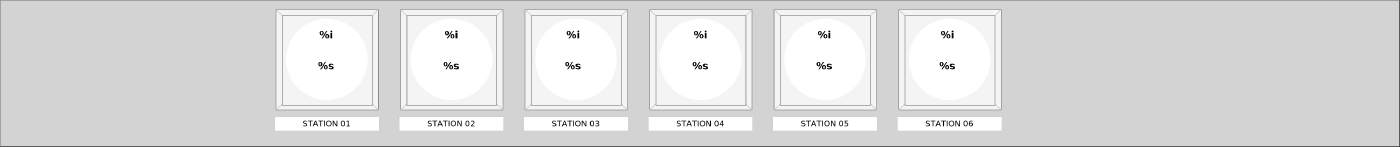
VISUALIZATION Popup_ProcessStatus  // 2001x211
    Rectangle (0,0 2001x211)
    Group (570,13 150x175)
        RoundedRectangle (0,154 150x21), "STATION 02"
        Image (2,0 147x145)
            p573394764: StartStop.Value
        Pie (11,9 129x129)
            p426801730: iDisplayTimeCycle[2]
            p2124672552: iDisplayTimeCycleEnd[2]
        Ellipse (17,14 116x116), colour toggle: bDisplayTimeCycleOn[2]
        Rectangle (29,42 92x79), "%s", text variable: ARsStnProcessName[2]
        Rectangle (41,22 69x30), "%i", text variable: ARiStnProcessTimeCD[2]
    Group (392,13 150x175)
        RoundedRectangle (0,154 150x21), "STATION 01"
        Image (2,0 147x145)
            p573394764: StartStop.Value
        Pie (11,9 129x129)
            p426801730: iDisplayTimeCycle[1]
            p2124672552: iDisplayTimeCycleEnd[1]
        Ellipse (17,14 116x116), colour toggle: bDisplayTimeCycleOn[1]
        Rectangle (28,42 92x79), "%s", text variable: ARsStnProcessName[1]
        Rectangle (40,22 69x30), "%i", text variable: ARiStnProcessTimeCD[1]
    Group (748,13 150x175)
        RoundedRectangle (0,154 150x21), "STATION 03"
        Image (2,0 147x145)
            p573394764: StartStop.Value
        Pie (11,9 129x129)
            p426801730: iDisplayTimeCycle[3]
            p2124672552: iDisplayTimeCycleEnd[3]
        Ellipse (17,14 116x116), colour toggle: bDisplayTimeCycleOn[3]
        Rectangle (25,42 92x79), "%s", text variable: ARsStnProcessName[3]
        Rectangle (37,22 69x30), "%i", text variable: ARiStnProcessTimeCD[3]
    Group (926,13 150x175)
        RoundedRectangle (0,154 150x21), "STATION 04"
        Image (2,0 147x145)
            p573394764: StartStop.Value
        Pie (11,9 129x129)
            p426801730: iDisplayTimeCycle[4]
            p2124672552: iDisplayTimeCycleEnd[4]
        Ellipse (17,14 116x116), colour toggle: bDisplayTimeCycleOn[4]
        Rectangle (29,42 92x79), "%s", text variable: ARsStnProcessName[4]
        Rectangle (41,22 69x30), "%i", text variable: ARiStnProcessTimeCD[4]
    Group (1104,13 150x175)
        RoundedRectangle (0,154 150x21), "STATION 05"
        Image (2,0 147x145)
            p573394764: StartStop.Value
        Pie (11,9 129x129)
            p426801730: iDisplayTimeCycle[5]
            p2124672552: iDisplayTimeCycleEnd[5]
        Ellipse (17,14 116x116), colour toggle: bDisplayTimeCycleOn[5]
        Rectangle (28,42 92x79), "%s", text variable: ARsStnProcessName[5]
        Rectangle (40,22 69x30), "%i", text variable: ARiStnProcessTimeCD[5]
    Group (1282,13 150x175)
        RoundedRectangle (0,154 150x21), "STATION 06"
        Image (2,0 147x145)
            p573394764: StartStop.Value
        Pie (11,9 129x129)
            p426801730: iDisplayTimeCycle[6]
            p2124672552: iDisplayTimeCycleEnd[6]
        Ellipse (17,14 116x116), colour toggle: bDisplayTimeCycleOn[6]
        Rectangle (26,42 92x79), "%s", text variable: ARsStnProcessName[6]
        Rectangle (38,22 69x30), "%i", text variable: ARiStnProcessTimeCD[6]
END_VISUALIZATION

(* stored: Version 1.1.0.1, ProductVersion 3.1.4024.12
   Visu Popup_ProcessStatus: Id {8f3313f7-cabf-4b7f-b708-3aabaabc5089} *)
